FUNCTION_BLOCK LINX215 (* Composite Function Block Type *)
  (* Standard: 61499-2 *)
  (* Version 1.0, 3/14/2024, linkwise-linn, LOYTEC electronics GmbH, template *)
  PACKAGE Main;
  {SET_ATTRIBUTE(Runtime.FBType.DPAL.Device, true)}
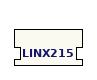
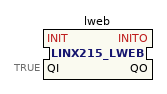
  FBS
    lweb : LINX215_LWEB(QI := TRUE);
  END_FBS
END_FUNCTION_BLOCK
